PROGRAM Axis05_Command
VAR
	Axis05: AXIS_REF;											//회전축
	Axis05_MC_Home: FB_HomeBeforeMoveAX8000;
	Axis05_MC_Power: MC_Power;
	Axis05_Status: MC_ReadStatus;
	Axis05_Position_Read: MC_ReadActualPosition;
	Axis05_Velocity_Read: MC_ReadActualVelocity;
	Axis05_Reset: MC_Reset;										//모터 알람 리셋
	Axis05_Stop: MC_Stop;										//모터 정지
	Axis05_Press_Move: MC_MoveAbsolute;
	Axis05_Home_Pos_Move: MC_MoveAbsolute;
	Axis05_Wait_Pos_Move: MC_MoveAbsolute;
	Axis05_Target_Pos_Move: MC_MoveAbsolute;
	Axis05_Work_End_Move: MC_MoveAbsolute;
	Axis05_Jog: MC_Jog;
	
	Always_ON	:	BOOL	:=TRUE	;//상시 ON
	Always_OFF	:	BOOL	:=FALSE	;//상시 OFF

	Home_Interlock			:	BOOL	;
	Home_Pos_Interlock		: 	BOOL	;
	Wait_Pos_Interlock		:	BOOL	;
	Target_Pos_Interlock	:	BOOL	;
	Work_End_POs_Interlock	:	BOOL	;
	Axis05_Calibration: MC_MoveAbsolute;
	Axis05_Maint_Move: MC_MoveAbsolute;
	Axis05_Tool_Change_Move: MC_MoveAbsolute;
	Axis05_Calibration_Move: MC_MoveAbsolute;
	Timer04: TON;
END_VAR
VAR // added by the converter: edge detectors and wires of the graphical bodies
    _rt1 : R_TRIG;
END_VAR

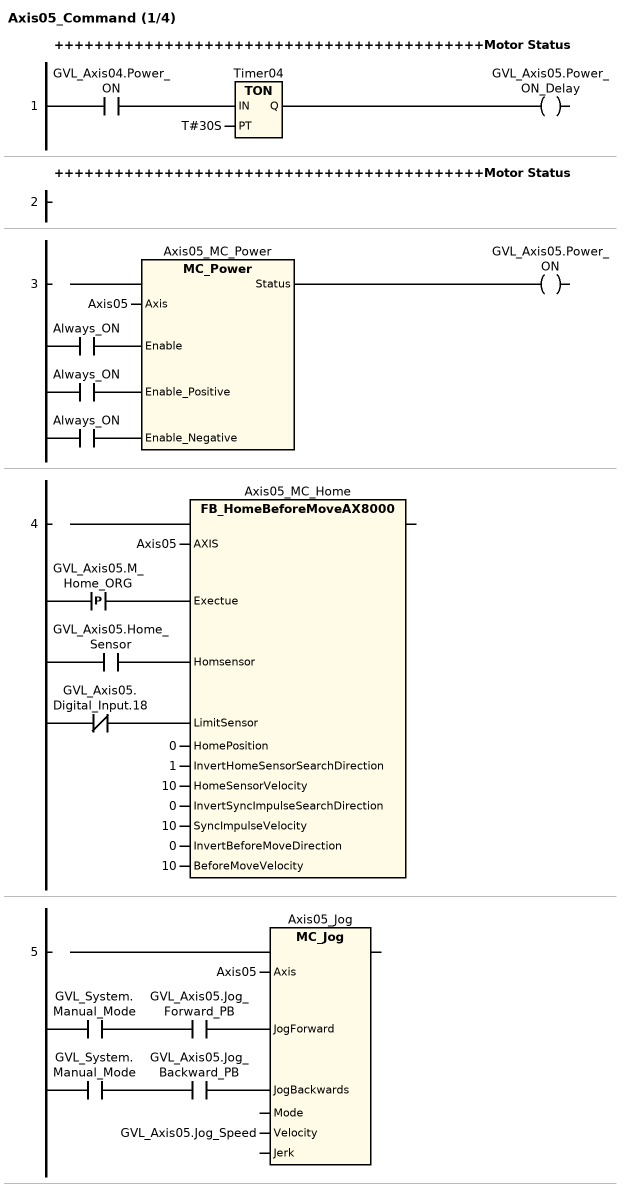
// NETWORK 1: +++++++++++++++++++++++++++++++++++++++++++Motor Status
Timer04(IN := GVL_Axis04.Power_ON, PT := T#30S); // TON
GVL_Axis05.Power_ON_Delay := Timer04.Q;

// NETWORK 2: +++++++++++++++++++++++++++++++++++++++++++Motor Status

// NETWORK 3
Axis05_MC_Power(
    Axis := Axis05,
    Enable := Always_ON,
    Enable_Positive := Always_ON,
    Enable_Negative := Always_ON); // MC_Power
GVL_Axis05.Power_ON := Axis05_MC_Power.Status;

// NETWORK 4
_rt1(CLK := GVL_Axis05.M_Home_ORG);
Axis05_MC_Home(
    AXIS := Axis05,
    Exectue := _rt1.Q,
    Homsensor := GVL_Axis05.Home_Sensor,
    LimitSensor := NOT GVL_Axis05.Digital_Input.18,
    HomePosition := 0,
    InvertHomeSensorSearchDirection := 1,
    HomeSensorVelocity := 10,
    InvertSyncImpulseSearchDirection := 0,
    SyncImpulseVelocity := 10,
    InvertBeforeMoveDirection := 0,
    BeforeMoveVelocity := 10); // FB_HomeBeforeMoveAX8000

// NETWORK 5
Axis05_Jog(
    Axis := Axis05,
    JogForward := GVL_System.Manual_Mode AND GVL_Axis05.Jog_Forward_PB,
    JogBackwards := GVL_System.Manual_Mode AND GVL_Axis05.Jog_Backward_PB,
    Velocity := GVL_Axis05.Jog_Speed); // MC_Jog

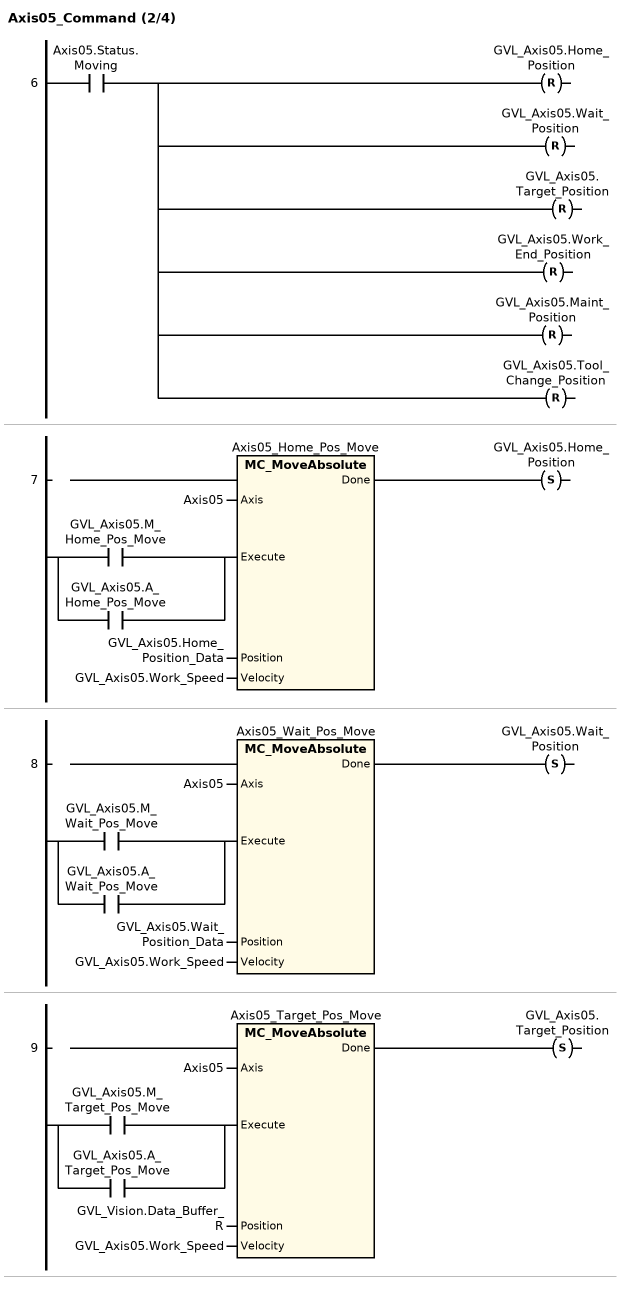
// NETWORK 6
GVL_Axis05.Home_Position R= Axis05.Status.Moving;
GVL_Axis05.Wait_Position R= Axis05.Status.Moving;
GVL_Axis05.Target_Position R= Axis05.Status.Moving;
GVL_Axis05.Work_End_Position R= Axis05.Status.Moving;
GVL_Axis05.Maint_Position R= Axis05.Status.Moving;
GVL_Axis05.Tool_Change_Position R= Axis05.Status.Moving;

// NETWORK 7
Axis05_Home_Pos_Move(
    Axis := Axis05,
    Execute := GVL_Axis05.M_Home_Pos_Move OR GVL_Axis05.A_Home_Pos_Move,
    Position := GVL_Axis05.Home_Position_Data,
    Velocity := GVL_Axis05.Work_Speed); // MC_MoveAbsolute
GVL_Axis05.Home_Position S= Axis05_Home_Pos_Move.Done;

// NETWORK 8
Axis05_Wait_Pos_Move(
    Axis := Axis05,
    Execute := GVL_Axis05.M_Wait_Pos_Move OR GVL_Axis05.A_Wait_Pos_Move,
    Position := GVL_Axis05.Wait_Position_Data,
    Velocity := GVL_Axis05.Work_Speed); // MC_MoveAbsolute
GVL_Axis05.Wait_Position S= Axis05_Wait_Pos_Move.Done;

// NETWORK 9
Axis05_Target_Pos_Move(
    Axis := Axis05,
    Execute := GVL_Axis05.M_Target_Pos_Move OR GVL_Axis05.A_Target_Pos_Move,
    Position := GVL_Vision.Data_Buffer_R,
    Velocity := GVL_Axis05.Work_Speed); // MC_MoveAbsolute
GVL_Axis05.Target_Position S= Axis05_Target_Pos_Move.Done;

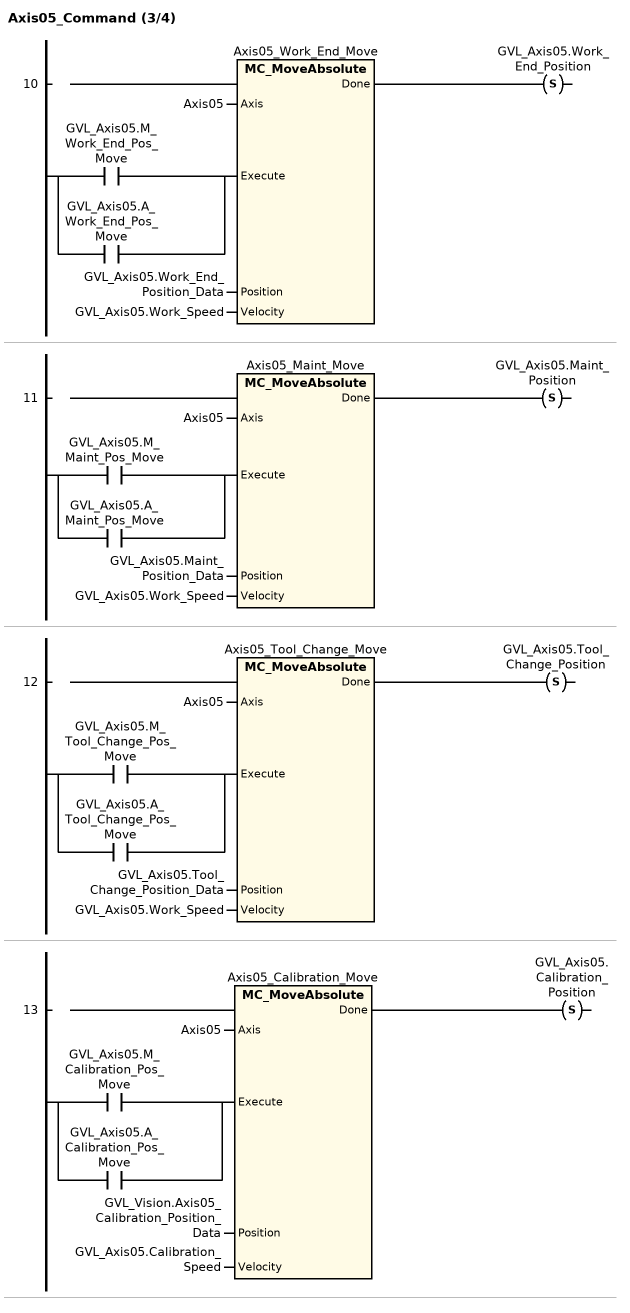
// NETWORK 10
Axis05_Work_End_Move(
    Axis := Axis05,
    Execute := GVL_Axis05.M_Work_End_Pos_Move OR GVL_Axis05.A_Work_End_Pos_Move,
    Position := GVL_Axis05.Work_End_Position_Data,
    Velocity := GVL_Axis05.Work_Speed); // MC_MoveAbsolute
GVL_Axis05.Work_End_Position S= Axis05_Work_End_Move.Done;

// NETWORK 11
Axis05_Maint_Move(
    Axis := Axis05,
    Execute := GVL_Axis05.M_Maint_Pos_Move OR GVL_Axis05.A_Maint_Pos_Move,
    Position := GVL_Axis05.Maint_Position_Data,
    Velocity := GVL_Axis05.Work_Speed); // MC_MoveAbsolute
GVL_Axis05.Maint_Position S= Axis05_Maint_Move.Done;

// NETWORK 12
Axis05_Tool_Change_Move(
    Axis := Axis05,
    Execute := GVL_Axis05.M_Tool_Change_Pos_Move OR GVL_Axis05.A_Tool_Change_Pos_Move,
    Position := GVL_Axis05.Tool_Change_Position_Data,
    Velocity := GVL_Axis05.Work_Speed); // MC_MoveAbsolute
GVL_Axis05.Tool_Change_Position S= Axis05_Tool_Change_Move.Done;

// NETWORK 13
Axis05_Calibration_Move(
    Axis := Axis05,
    Execute := GVL_Axis05.M_Calibration_Pos_Move OR GVL_Axis05.A_Calibration_Pos_Move,
    Position := GVL_Vision.Axis05_Calibration_Position_Data,
    Velocity := GVL_Axis05.Calibration_Speed); // MC_MoveAbsolute
GVL_Axis05.Calibration_Position S= Axis05_Calibration_Move.Done;

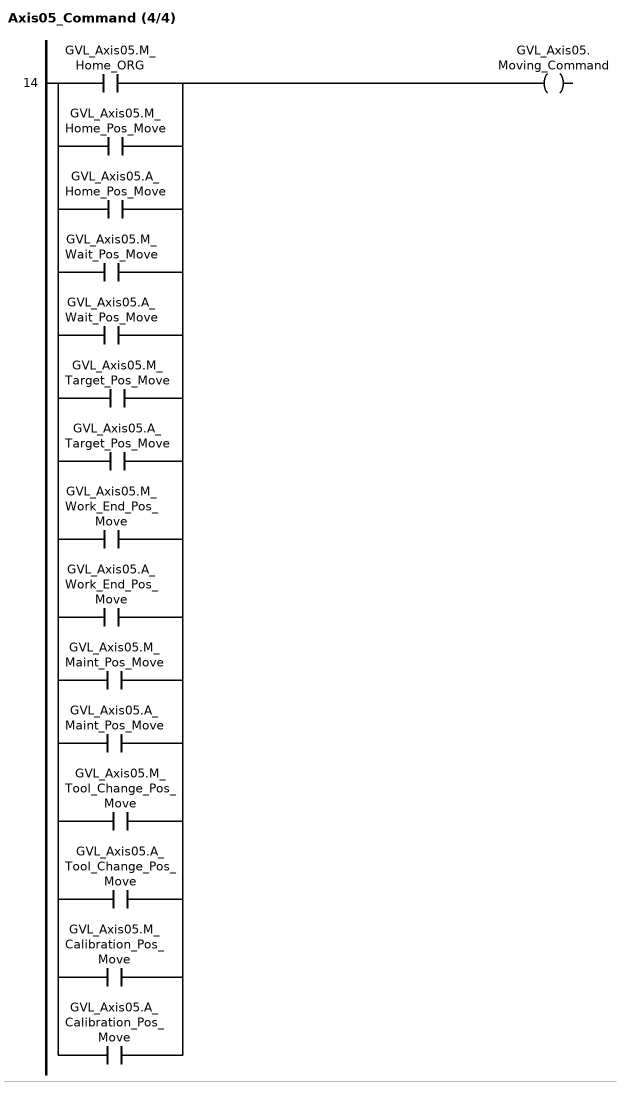
// NETWORK 14
GVL_Axis05.Moving_Command := GVL_Axis05.M_Home_ORG OR GVL_Axis05.M_Home_Pos_Move OR GVL_Axis05.A_Home_Pos_Move OR GVL_Axis05.M_Wait_Pos_Move OR GVL_Axis05.A_Wait_Pos_Move OR GVL_Axis05.M_Target_Pos_Move OR GVL_Axis05.A_Target_Pos_Move OR GVL_Axis05.M_Work_End_Pos_Move OR GVL_Axis05.A_Work_End_Pos_Move OR GVL_Axis05.M_Maint_Pos_Move OR GVL_Axis05.A_Maint_Pos_Move OR GVL_Axis05.M_Tool_Change_Pos_Move OR GVL_Axis05.A_Tool_Change_Pos_Move OR GVL_Axis05.M_Calibration_Pos_Move OR GVL_Axis05.A_Calibration_Pos_Move;

END_PROGRAM

(* stored: Version 1.1.0.1, ProductVersion 3.1.4024.15
   POU Axis05_Command: Id {4d1dcb0d-bbba-42ea-8a19-f6e44966261c}, SpecialFunc None *)
